# EPICS substitutions: es2-eps/es2-epsApp/Db/es2-eps-misc.substitutions
file plc1-misc-di.template
{
        pattern { Sys		, Dev			, PLC		}
		{ XF:23ID2-ES	, "{APPES_LL-LSw:1}"	, XF23ID2_EPS	}
		{ XF:23ID2-ES	, "{IOXAS_LL-LSw:1}"	, XF23ID2_EPS	}
		{ XF:23ID2-ES   , "{IOXAS_LL-LSw:1}"	, XF23ID2_EPS   }
}
